(* PLC project P1AM Function Blocks, OpenPLC P1AM Function Blocks Library 1.0, author Thiago Alves *)
(* stored: creationDateTime 2021-11-11T02:33:11, modificationDateTime 2021-11-11T02:33:11 *)

(* This block outputs the sum of input I0 and 10. *)
FUNCTION_BLOCK Test
  VAR_INPUT
    I0 : INT;  (* Insert an integer here *)
    ACTIVE : BOOL;  (* 0 – block does nothing, 1 – block sums 10 to integer in I0 *)
  END_VAR
  VAR_OUTPUT
    OUT : INT;  (* This is the output: I0 + 10 *)
  END_VAR

						
							
						
					
END_FUNCTION_BLOCK
